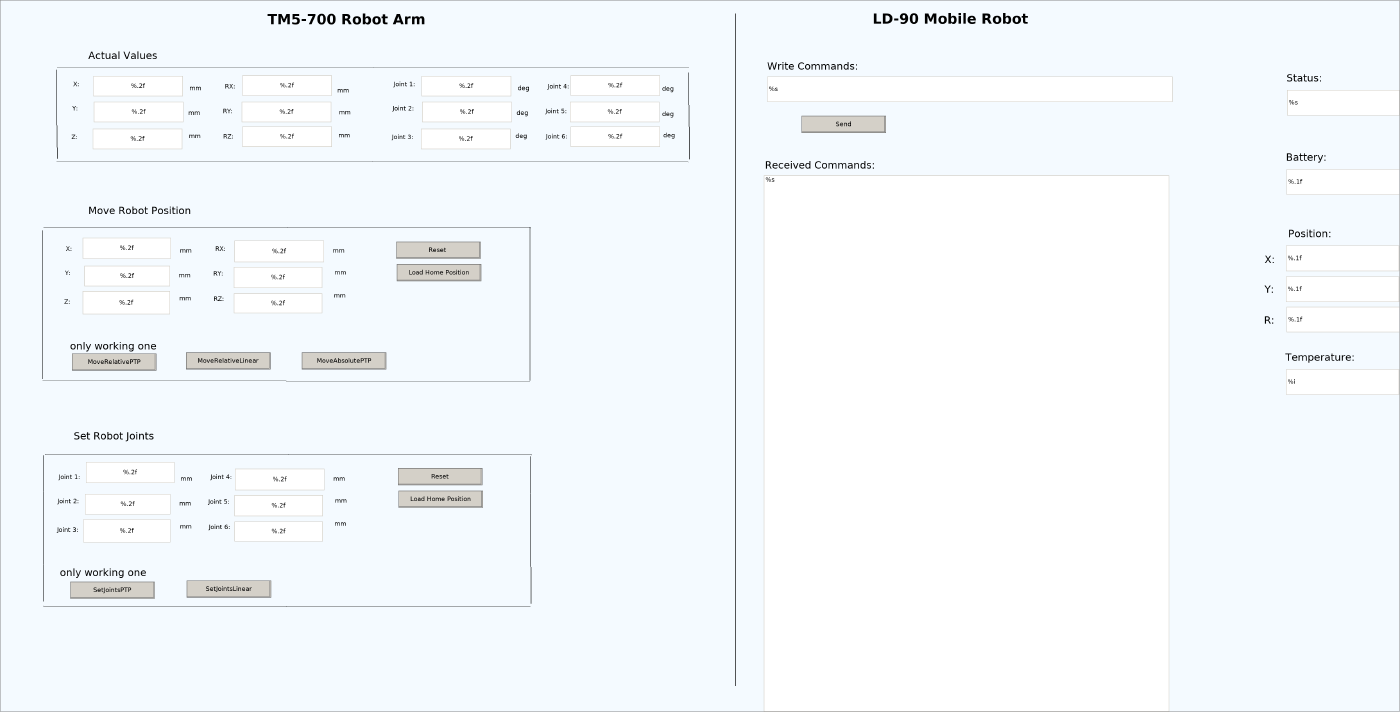
VISUALIZATION CommandWindow  // 2491x1267
    Textfield (147,423 157x37), "%.2f", text variable: GVL_CommandWindow.fX_Ref
        OnMouseClick: write the text variable via Default
    Textfield (150,473 152x36), "%.2f", text variable: GVL_CommandWindow.fY_Ref
        OnMouseClick: write the text variable via Default
    Textfield (147,518 155x41), "%.2f", text variable: GVL_CommandWindow.fZ_Ref
        OnMouseClick: write the text variable via Default
    Textfield (417,428 159x38), "%.2f", text variable: GVL_CommandWindow.fRX_Ref
        OnMouseClick: write the text variable via Default
    Textfield (416,475 157x37), "%.2f", text variable: GVL_CommandWindow.fRY_Ref
        OnMouseClick: write the text variable via Default
    Textfield (416,522 157x35), "%.2f", text variable: GVL_CommandWindow.fRZ_Ref
        OnMouseClick: write the text variable via Default
    Textfield (166,135 159x36), "%.2f", text variable: GVL_MobileManipulator.stRobotArmObjectTM.fX
    Textfield (167,181 159x36), "%.2f", text variable: GVL_MobileManipulator.stRobotArmObjectTM.fY
    Textfield (165,229 159x36), "%.2f", text variable: GVL_MobileManipulator.stRobotArmObjectTM.fZ
    Textfield (431,134 159x36), "%.2f", text variable: GVL_CommandWindow.fRX_Current
    Textfield (430,181 159x36), "%.2f", text variable: GVL_MobileManipulator.stRobotArmObjectTM.fRY
    Textfield (431,225 159x36), "%.2f", text variable: GVL_MobileManipulator.stRobotArmObjectTM.fRZ
    Label (109,133 53x34), "X:"
    Label (107,176 53x34), "Y:"
    Label (106,227 53x34), "Z:"
    Label (383,137 53x34), "RX:"
    Label (379,181 53x34), "RY:"
    Label (380,226 53x34), "RZ:"
    Label (334,142 40x30), "mm"
    Label (332,186 40x30), "mm"
    Label (333,227 40x30), "mm"
    Label (597,146 40x30), "mm"
    Label (600,185 40x30), "mm"
    Label (599,226 40x30), "mm"
    Label (85,82 273x34), "Actual Values"
    Label (83,358 331x34), "Move Robot Position"
    Textfield (750,135 159x36), "%.2f", text variable: GVL_MobileManipulator.stRobotArmObjectTM.fTheta1
    Textfield (751,181 159x36), "%.2f", text variable: GVL_MobileManipulator.stRobotArmObjectTM.fTheta2
    Textfield (749,229 159x36), "%.2f", text variable: GVL_MobileManipulator.stRobotArmObjectTM.fTheta3
    Textfield (1015,134 159x36), "%.2f", text variable: GVL_MobileManipulator.stRobotArmObjectTM.fTheta4
    Textfield (1014,181 159x36), "%.2f", text variable: GVL_MobileManipulator.stRobotArmObjectTM.fTheta5
    Textfield (1015,225 159x36), "%.2f", text variable: GVL_MobileManipulator.stRobotArmObjectTM.fTheta6
    Label (693,133 53x34), "Joint 1:"
    Label (691,176 53x34), "Joint 2:"
    Label (690,227 53x34), "Joint 3:"
    Label (967,137 53x34), "Joint 4:"
    Label (963,181 53x34), "Joint 5:"
    Label (964,226 53x34), "Joint 6:"
    Label (918,142 40x30), "deg"
    Label (916,186 40x30), "deg"
    Label (914,227 40x30), "deg"
    Label (1175,143 40x30), "deg"
    Label (1175,188 40x30), "deg"
    Label (1177,226 40x30), "deg"
    Label (96,426 53x34), "X:"
    Label (94,469 53x34), "Y:"
    Label (93,520 53x34), "Z:"
    Label (366,426 53x34), "RX:"
    Label (362,470 53x34), "RY:"
    Label (363,515 53x34), "RZ:"
    Label (317,431 40x30), "mm"
    Label (315,475 40x30), "mm"
    Label (316,516 40x30), "mm"
    Label (589,431 40x30), "mm"
    Label (592,470 40x30), "mm"
    Label (591,511 40x30), "mm"
    Button (128,629 150x30), "MoveRelativePTP"
        tap GVL_CommandWindow.bCmdMoveRelPTP
        OnMouseClick: execute { GVL_CommandWindow.commandID := MoveCartesianPTP; }
    Button (331,627 150x30), "MoveRelativeLinear"
        tap GVL_CommandWindow.bCmdMoveRelLinear
        OnMouseClick: execute { GVL_CommandWindow.commandID := MoveCartesianLine; }
    Button (537,627 150x30), "MoveAbsolutePTP"
    Button (706,470 150x30), "Load Home Position"
        OnMouseClick: execute {
            GVL_CommandWindow.fX_Ref := 100;
            GVL_CommandWindow.fY_Ref := 100;
            GVL_CommandWindow.fZ_Ref := 100;
            GVL_CommandWindow.fRX_Ref := 0;
            GVL_CommandWindow.fRY_Ref := 0;
            GVL_CommandWindow.fRZ_Ref := 90;
        }
    Textfield (153,822 157x37), "%.2f", text variable: GVL_CommandWindow.fTheta1_Ref
        OnMouseClick: write the text variable via Default
    Textfield (151,879 152x36), "%.2f", text variable: GVL_CommandWindow.fTheta2_Ref
        OnMouseClick: write the text variable via Default
    Textfield (148,924 155x41), "%.2f", text variable: GVL_CommandWindow.fTheta3_Ref
        OnMouseClick: write the text variable via Default
    Textfield (418,834 159x38), "%.2f", text variable: GVL_CommandWindow.fTheta4_Ref
        OnMouseClick: write the text variable via Default
    Textfield (417,881 157x37), "%.2f", text variable: GVL_CommandWindow.fTheta5_Ref
        OnMouseClick: write the text variable via Default
    Textfield (417,928 157x35), "%.2f", text variable: GVL_CommandWindow.fRZ_Ref
        OnMouseClick: write the text variable via Default
    Label (97,832 53x34), "Joint 1:"
    Label (95,875 53x34), "Joint 2:"
    Label (94,926 53x34), "Joint 3:"
    Label (367,832 53x34), "Joint 4:"
    Label (363,876 53x34), "Joint 5:"
    Label (364,921 53x34), "Joint 6:"
    Label (318,837 40x30), "mm"
    Label (316,881 40x30), "mm"
    Label (317,922 40x30), "mm"
    Label (590,837 40x30), "mm"
    Label (593,876 40x30), "mm"
    Label (592,917 40x30), "mm"
    Button (125,1035 150x30), "SetJointsPTP"
        tap GVL_CommandWindow.bCmdSetJointsPTP
        OnMouseClick: execute { GVL_CommandWindow.commandID := SetJointPositions; }
    Button (332,1033 150x30), "SetJointsLinear"
    Button (708,833 150x30), "Reset"
        OnMouseClick: execute {
            GVL_CommandWindow.fTheta1_Ref := 0;
            GVL_CommandWindow.fTheta2_Ref := 0;
            GVL_CommandWindow.fTheta3_Ref := 0;
            GVL_CommandWindow.fTheta4_Ref := 0;
            GVL_CommandWindow.fTheta5_Ref := 0;
            GVL_CommandWindow.fTheta6_Ref := 0;
        }
    Label (37,759 331x34), "Set Robot Joints"
    Button (705,430 150x30), "Reset"
        OnMouseClick: execute {
            GVL_CommandWindow.fX_Ref := 0;
            GVL_CommandWindow.fY_Ref := 0;
            GVL_CommandWindow.fZ_Ref := 0;
            GVL_CommandWindow.fRX_Ref := 0;
            GVL_CommandWindow.fRY_Ref := 0;
            GVL_CommandWindow.fRZ_Ref := 0;
        }
    Button (709,873 150x30), "Load Home Position"
        OnMouseClick: execute {
            GVL_CommandWindow.fTheta1_Ref := 0;
            GVL_CommandWindow.fTheta2_Ref := 90;
            GVL_CommandWindow.fTheta3_Ref := 0;
            GVL_CommandWindow.fTheta4_Ref := 0;
            GVL_CommandWindow.fTheta5_Ref := 0;
            GVL_CommandWindow.fTheta6_Ref := 0;
        }
    Label (36,599 331x34), "only working one"
    Label (18,1002 331x34), "only working one"
    Textfield (1359,312 721x955), "%s", text variable: GVL_CommandWindow.sReceivedCommands
    Label (1358,279 252x30), "Received Commands:"
    Textfield (1365,136 721x45), "%s", text variable: GVL_CommandWindow.sWriteCommand
        OnMouseClick: write the text variable via Default
    Label (1362,103 219x30), "Write Commands:"
    Button (1426,206 150x30), "Send"
        tap GVL_CommandWindow.bCmdWriteStringToLD90
    Line (101,287) (1224,288)
    Line (1309,1220) (1309,24)
    Line (1227,283) (1225,129)
    Line (102,119) (1225,120)
    Line (102,282) (100,124)
    Label (480,17 273x34), "TM5-700 Robot Arm"
    Label (1555,16 273x34), "LD-90 Mobile Robot"
    Line (76,674) (76,410)
    Line (76,677) (942,678)
    Line (78,404) (944,405)
    Line (80,808) (946,809)
    Line (77,1078) (943,1079)
    Line (943,677) (943,404)
    Line (78,1070) (77,810)
    Line (945,1074) (944,812)
    Textfield (2290,160 201x45), "%s", text variable: GVL_MobileManipulator.stMobileRobotObjectLD.sStatus
        OnMouseClick: write the text variable via Default
    Label (2286,124 117x30), "Status:"
    Textfield (2289,301 201x45), "%.1f", text variable: GVL_MobileManipulator.stMobileRobotObjectLD.fBattery
        OnMouseClick: write the text variable via Default
    Label (2285,265 117x30), "Battery:"
    Textfield (2288,437 201x45), "%.1f", text variable: GVL_MobileManipulator.stMobileRobotObjectLD.fPositionX
        OnMouseClick: write the text variable via Default
    Label (2289,401 117x30), "Position:"
    Textfield (2288,492 201x45), "%.1f", text variable: GVL_MobileManipulator.stMobileRobotObjectLD.fPositionY
        OnMouseClick: write the text variable via Default
    Textfield (2289,546 201x45), "%.1f", text variable: GVL_MobileManipulator.stMobileRobotObjectLD.fRotationTheta
        OnMouseClick: write the text variable via Default
    Textfield (2288,657 201x45), "%i", text variable: GVL_MobileManipulator.stMobileRobotObjectLD.nTemperature
        OnMouseClick: write the text variable via Default
    Label (2284,621 117x30), "Temperature:"
    Label (2247,447 28x30), "X:"
    Label (2247,500 28x30), "Y:"
    Label (2246,555 28x30), "R:"
END_VISUALIZATION

(* stored: Version 1.1.0.1, ProductVersion 3.1.4024.11
   Visu CommandWindow: Id {5bada566-9073-4cf6-93ef-39466ba07087} *)
